FUNCTION_BLOCK Test_ListClear EXTENDS T_UnitTestBase
VAR
    List  : T_ListOfTests(Capacity := 10);
    Test0 : Test_ExampleTest;
    Test1 : Test_ExampleTest;
    Test2 : Test_ExampleTest;
    Test3 : Test_ExampleTest;
END_VAR

METHOD Init
SUPER^.Init();
List.Clear();
List.AddTest(Test0);
List.AddTest(Test1);
List.AddTest(Test2);
List.AddTest(Test3);
END_METHOD

METHOD RunTest
AssertIsTrue(Condition := List.Count = 4,
             Message   := 'List.Count was not 4');
			 
List.Clear();			 

AssertIsTrue(Condition := List.Count = 0,
             Message   := 'List.Count was not 0');

TestCompleted := TRUE;
END_METHOD

END_FUNCTION_BLOCK

(* stored: Version 1.1.0.1, ProductVersion 3.1.4024.12
   POU Test_ListClear: Id {99e29a87-ac8b-4ed1-8471-2846d4f2813c}, SpecialFunc None
   Method Init: Id {8a021792-fedf-418c-9fa3-308d88b77576}
   Method RunTest: Id {4404b0c7-fb1a-449c-948d-c29a698c43db} *)
